FUNCTION_BLOCK FINAL FB_MoveA EXTENDS FB_StatusExecuteFB IMPLEMENTS ITF_ExtendsFB
VAR_IN_OUT
	fbMover								: MC_PlanarMover;
END_VAR
VAR_INPUT
	Execute								: BOOL;
	Position							: DUT_Position;
	Velocity							: LREAL;
	Acceleration						: LREAL;
	Deceleration						: LREAL;
	Jerk								: LREAL;
END_VAR
VAR_OUTPUT
	Done								: BOOL;
	Busy								: BOOL;
	CommandAborted						: BOOL;
	Error								: BOOL;
	ErrorID								: UDINT;
END_VAR
VAR
	uiState								: UINT;
	//Input 内部変数
	dutPosition							: DUT_Position;
	lrVelocity							: LREAL;
	lrAcceleration						: LREAL;
	lrDeceleration						: LREAL;
	lrJerk								: LREAL;
	
	//ローカル
	fbFB_Mover							: MC_PlanarFeedback;
	fbConstraint						: DynamicConstraint_PathXY;
END_VAR

Prop_Execute := Execute;
METH_Main();

fbFB_Mover.Update();

Busy := bBusy;
Done := bDone;
CommandAborted := bCommandAborted;
Error := bError;
ErrorID := udiErrorID;

//{error 'add method implementation or delete method to use base implementation'}
METHOD METH_Busy : BOOL
IF fbFB_Mover.Error THEN
	METH_Error();
	Prop_ErrorID := fbFB_Mover.ErrorId; //Moverがエラー
	RETURN;
END_IF
IF THIS^.fbMover.MCTOPLC.STD.State = MC_PLANAR_STATE.Error THEN
	METH_Error();
	Prop_ErrorID := 1; //Moverがエラー
	RETURN;
END_IF
IF fbFB_Mover.Aborted THEN
	METH_CommandAborted();
	RETURN;
END_IF

CASE THIS^.uiState OF
	0:
	fbConstraint.SetValuesVADJ(V:= THIS^.lrVelocity, A:= THIS^.lrAcceleration, D:= THIS^.lrDeceleration, J:= THIS^.lrJerk);
	THIS^.fbMover.MoveA(
		commandFeedback:= THIS^.fbFB_Mover, 
		targetPosition:= dutPosition.a, 
		constraint:= fbConstraint);

	THIS^.uiState := 10;	
	
	10:
	IF fbFB_Mover.Done THEN
		THIS^.uiState := 16#FFFF;	
	END_IF
	
	16#FFFF:
	METH_Done();
END_CASE
END_METHOD

//{error 'add method implementation or delete method to use base implementation'}
METHOD METH_Enter : BOOL
//Input 内部変数に移す
dutPosition := Position;
lrVelocity := Velocity;
lrAcceleration := Acceleration;
lrDeceleration := Deceleration;
lrJerk := Jerk;
END_METHOD

//{error 'add method implementation or delete method to use base implementation'}
METHOD METH_Exit : BOOL
Prop_Done := FALSE;
Prop_Busy := FALSE;
Prop_CommandAborted := FALSE;
Prop_Error := FALSE;
Prop_ErrorID := 0;

// 内部変数をリフレッシュする
uiState := 0;
lrVelocity := 0;
lrAcceleration := 0;
lrDeceleration := 0;
lrJerk := 0;
END_METHOD

//{error 'add method implementation or delete method to use base implementation'}
METHOD METH_Main : BOOL
//Doneに遷移
IF SUPER^.bDone AND SUPER^.bExecute THEN
	METH_Done();
	RETURN;
END_IF
//Errorに遷移
IF SUPER^.bError AND SUPER^.bExecute THEN
	METH_Error();
	RETURN;
END_IF
//CommandAbortedに遷移
IF SUPER^.bCommandAborted AND SUPER^.bExecute THEN
	METH_CommandAborted();
	RETURN;
END_IF
//FBをリフレッシュ
//状態がDone, Error, CommandAborted時に Execute FALSE で遷移
IF (SUPER^.bDone OR SUPER^.bError OR SUPER^.bCommandAborted) AND NOT SUPER^.bExecute THEN
	METH_Exit();
	RETURN;
END_IF

//実行開始
IF SUPER^.bExecute AND NOT SUPER^.bBusy THEN
	METH_Execute();
	METH_Enter();
END_IF
//実行中
IF SUPER^.bBusy THEN
	METH_Busy();
END_IF
END_METHOD

END_FUNCTION_BLOCK

(* stored: Version 1.1.0.1, ProductVersion 3.1.4024.11
   POU FB_MoveA: Id {4cb3418a-78dc-4390-9ab8-6839788d286c}, SpecialFunc None
   Method METH_Busy: Id {3b9d7e17-f7be-4e3a-88ef-330da940cc02}
   Method METH_Enter: Id {a2bccc4f-0c37-4c75-81b7-a668f6bf5e28}
   Method METH_Exit: Id {5b6c1e73-c1ad-41f0-94bd-cba02e0c757d}
   Method METH_Main: Id {8ddadc5e-718c-45c1-844a-e1556fb58719} *)
